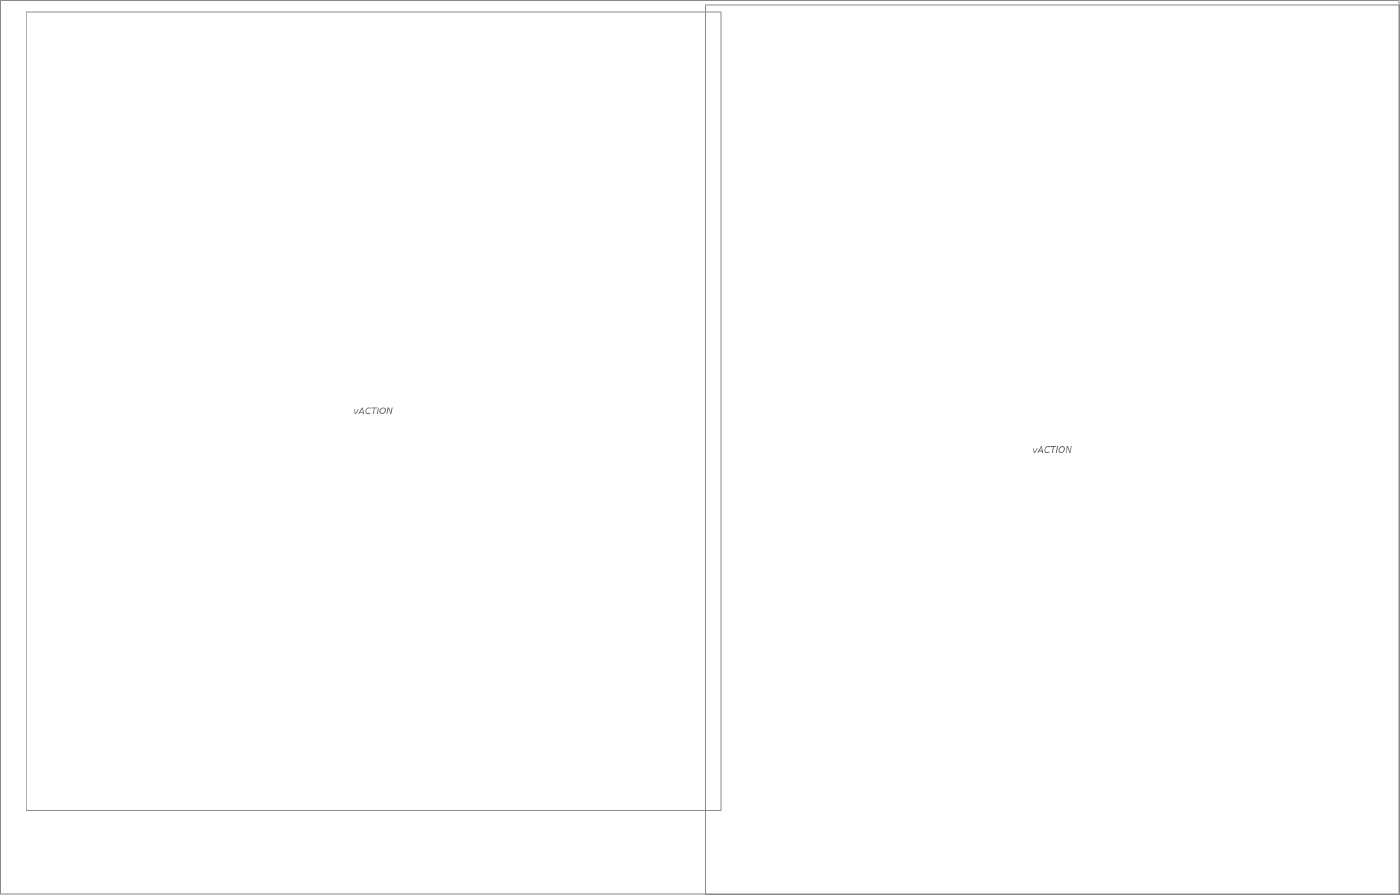
VISUALIZATION Visualization  // 1571x1005
    Frame (29,13 780x897)
        shows vACTION(vACTION := ACTION1)
    Frame (791,5 780x1000)
        shows vACTION(vACTION := ACTION2)
END_VISUALIZATION

(* stored: Version 1.1.0.1, ProductVersion 3.1.4024.12
   Visu Visualization: Id {4537162b-5f0d-49cf-ad43-cab00bff90cc} *)
